TYPE ST_DataPntAdr :
STRUCT
	pAddress		:UDINT;
	udiSize		:UDINT;
END_STRUCT
END_TYPE

(* stored: Version 1.1.0.1
   DUT ST_DataPntAdr: Id {72a74ecb-35c4-4719-bd55-6136aa6217d9} *)
